FUNCTION_BLOCK FB_TcMessageSuccess EXTENDS FB_TcMessage
VAR
END_VAR

METHOD FB_init : BOOL
VAR_INPUT
	bInitRetains: BOOL; // if TRUE, the retain variables are initialized (warm start / cold start)
	bInCopyCode: BOOL; // if TRUE, the instance afterwards gets moved into the copy code (online change)
END_VAR
VAR
END_VAR
IF NOT bInCopyCode THEN
	SUPER^.CreateEx(Tc3_EventLogger.SUCCESS_EVENT, 0);
END_IF
END_METHOD

END_FUNCTION_BLOCK

(* stored: POU FB_TcMessageSuccess: Id 764f8c59-3664-4a1d-a4d1-dcd3533d3b46, SpecialFunc None
   Method FB_init: Id b71f0de6-2b15-4b45-926a-02c488256cdb *)
